PROGRAM prg_Druktoets_Functies
VAR
END_VAR

END_PROGRAM

(* stored: Version 1.1.0.1, ProductVersion 3.1.4024.15
   POU prg_Druktoets_Functies: Id {b8b4c91c-3c6c-45af-bdd6-4f5f22eeb854}, SpecialFunc None *)
